(* PLC project LD_EVOLUTION_1, Beckhoff Automation GmbH TwinCAT PLC Control 3.5.10.30 *)
(* stored: creationDateTime 2019-09-26T16:12:41.2429215, modificationDateTime 2019-09-26T16:12:41.2429215 *)

PROGRAM Main
VAR
	A: BOOL;
	B: BOOL;
	Open: BOOL;
END_VAR

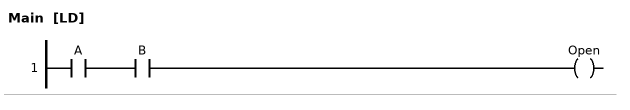
(* LD diagram, written out as Structured Text *)

Open := A AND B;
END_PROGRAM

CONFIGURATION Application
  RESOURCE LD_EVOLUTION_1 ON PLC
    TASK PlcTask(INTERVAL := T#0ms, PRIORITY := 20);
    PROGRAM Main WITH PlcTask : Main;
  END_RESOURCE
END_CONFIGURATION
